PROGRAM P_API_IO
VAR
END_VAR

gvl_api.stAxis[FastScan].Origin:=Axis[FastScan].IO.snHome;
gvl_api.stAxis[FastScan].LimitP:=Axis[FastScan].IO.snLimitP;
gvl_api.stAxis[Z_Axis].Origin:=Axis[Z_Axis].IO.snHome;
gvl_api.stAxis[Z_Axis].LimitP:=Axis[Z_Axis].IO.snLimitP;

END_PROGRAM

(* stored: Version 1.1.0.1, ProductVersion 3.1.4024.11
   POU P_API_IO: Id {120f89c6-aa84-4ed3-9662-362dea3b6d11}, SpecialFunc None *)
